FUNCTION_BLOCK NodeProtectionExtension EXTENDS ExtensionBase IMPLEMENTS I_EventHandler
VAR
	parent : I_NodeWithProtection;
	nodeProperty_Protection : Parameter('protection','BOOL', THIS^);
END_VAR

METHOD FB_exit : BOOL
VAR_INPUT
	bInCopyCode : BOOL; // if TRUE, the exit method is called for exiting an instance that is copied afterwards (online change).
END_VAR
IF bInCopyCode THEN
	RETURN;
END_IF

UnregisterWithParent();
END_METHOD

METHOD FB_init : BOOL
VAR_INPUT
	bInitRetains : BOOL; // if TRUE, the retain variables are initialized (warm start / cold start)
	bInCopyCode : BOOL;  // if TRUE, the instance afterwards gets moved into the copy code (online change)
	Name : T_MAXSTRING;
	Parent : I_NodeWithProtection;
END_VAR
THIS^.parent := Parent;
RegisterWithParent();
END_METHOD

METHOD PUBLIC HandleEvent
VAR_INPUT
	Event : I_Event;
END_VAR
VAR
	nodePreExecuteEvent : I_NodePreExecuteEvent;
	preExecuteResult : HRESULT;
END_VAR
IF NOT __QUERYINTERFACE(Event, nodePreExecuteEvent) THEN
	RETURN;
END_IF

IF nodePreExecuteEvent.ExecuteCancelled THEN 
	RETURN;
END_IF

IF NOT IsProtected THEN
	RETURN;
END_IF

preExecuteResult := parent.PreExecuteCheck();

IF SUCCEEDED(preExecuteResult) THEN
	RETURN;
END_IF

nodePreExecuteEvent.Cancel();
END_METHOD

PROPERTY PUBLIC IsProtected : BOOL
GET
VAR
	value : BOOL;
END_VAR
nodeProperty_Protection.TryGet(value);
IsProtected := value;
END_GET
END_PROPERTY

METHOD PROTECTED RegisterWithParent
VAR_INPUT
END_VAR
IF parent = 0 THEN
	RETURN;
END_IF

parent.AddExtension(THIS^);
parent.OnEvent('OnNodePreExecute',THIS^);
END_METHOD

METHOD PROTECTED UnregisterWithParent
VAR_INPUT
END_VAR
IF parent = 0 THEN
	RETURN;
END_IF

parent.OffEvent('OnNodePreExecute',THIS^);
END_METHOD

END_FUNCTION_BLOCK

(* stored: Version 1.1.0.1, ProductVersion 3.1.4024.12
   POU NodeProtectionExtension: Id {9333f4ac-bf14-0883-31a3-a1646eee6f26}, SpecialFunc None
   Folder Constructor: Id {5ef21104-2841-0bc0-09ab-332c7665e59d}
   Folder Destructor: Id {74c6b421-49ed-0857-3dc1-3488abf310fc}
   Folder Protected: Id {56670b6a-e74a-0d02-3a94-42080bcf64ac}
   Method FB_exit: Id {17033b86-661f-0c7f-3f6d-1e18005f3e47}
   Method FB_init: Id {3f82d6c4-7348-0f4e-330a-7f09298b6602}
   Method HandleEvent: Id {947efc4f-860b-0b89-31c7-ed2e9660491d}
   Property IsProtected: Id {36f6679e-b7ee-0abf-0b5e-78fa56990537}
   Get Get: Id {c975c975-d4c4-0b40-278e-a6e0ae19b99a}
   Method RegisterWithParent: Id {8d0d5853-572c-0a01-0c9a-3689592ed625}
   Method UnregisterWithParent: Id {d1a8c63a-75ba-0f55-3e18-bd204f36815e} *)
